(* CoDeSys 2.3.9.31 project: Test4(7Axis).pro *)
(* Libraries: STANDARD.LIB 5.6.98 11:03:02 *)

(* Task configuration *)
TASK Standard (PRIORITY := 0, INTERVAL := T#10ms);
	MAIN
END_TASK

(* Global variable list: Global_Variables *)
VAR_GLOBAL
(**DB Address**)
	DB8 AT %MW2010:ARRAY[0..100] OF INT;
(*******用到的数组值有以下变量*******)

	CigMakingSpeed  AT %IW330:INT;
(**Packer Address Define**)
	PackingSpeed  AT %IW332:INT;
(*ManPotentiometerSpeed  Address*)
	PotenSpeed AT %IW328:INT;
(*****Level Address  Define********)
	ElevatorLevel AT %IW324:INT;
(*****Drop Address  Define********)
	DropLevel AT %IW326:INT;

	Store_set_zero AT %MX1000.0 : BOOL;
	test_run AT %MX1000.6 : BOOL;
	StoreUnit_discharge_button AT %MX2603.6 : BOOL;
	Elevater_man_paikong AT %MX2603.7 :BOOL;
	test_run_unprotected AT %MX1000.7 : BOOL;
	test_maker_speed AT %MW1950 : INT;
	test_packer_speed AT %MW1952 : INT;
	Corner_manual_speed AT %MW254 : INT;
	Store_manual_speed AT %MW260 : INT;
	DropTrans_cig_speed AT %MW2320 : INT;(*下降口输送烟支速度*)(*******7Axis**********)
	DropTrans_speed_rpm AT %MW2340 : INT;(*下降口输送电机转速*)(******7Axis***********)


	Lift_p_parameter AT %MW270 : INT;
	Transfer_p_parameter AT %MW272 : INT;
	MakerExport_p_parameter AT %MW274 : INT;



	Emergency_stop AT %IX0.0:BOOL;(*紧急停止继电器*)
	MakerExit_power AT %IX0.1:BOOL;(*备用*)
	Sample_power AT %IX0.2:BOOL;(*取样伺服主电源*)
	Corner_power AT %IX0.3:BOOL;(*弯道伺服主电源*)
	Lift_power AT %IX0.4:BOOL;(*提升伺服主电源*)
	Transfer_power AT %IX0.5:BOOL;(*传送伺服主电源*)
	Slope_power AT %IX0.6:BOOL;(*斜向伺服主电源*)
	Store_power AT %IX0.7:BOOL;(*存储伺服主电源*)
	DropTrans_power AT %IX1.0:BOOL;(*下降口输送伺服主电源*)(****************************************************7Axis中用DropTrans_power替换原Spare10*************)

	Spare11 AT %IX1.1:BOOL;(*备用*)
	MakerExit_servo_fault AT %IX1.2:BOOL;(*备用*)
	Sample_servo_fault AT %IX1.3:BOOL;(*取样伺服控制器故障*)
	Corner_servo_fault AT %IX1.4:BOOL;(*弯道伺服控制器故障*)
	Lift_servo_fault AT %IX1.5:BOOL;(*提升伺服控制器故障*)
	Transfer_servo_fault AT %IX1.6:BOOL;(*传送伺服控制器故障*)
	Slope_servo_fault AT %IX1.7:BOOL;(*斜向伺服控制器故障*)
	Store_servo_fault AT %IX2.0:BOOL;(*存储伺服控制器故障*)
	DropTrans_servo_fault AT %IX2.1:BOOL;(*备用*)(********************************************************************7Axis中用DropTrans_servo_fault替换原Spare21*************)
	Spare22 AT %IX2.2:BOOL;(*备用*)
	Elevater_man_auto_sw AT %IX2.3:BOOL;(*备用*)
	Elevater_start_pb AT %IX2.4:BOOL;(*备用*)
	DropTransLowLevel AT %IX2.5:BOOL;(*下降口输送低料位*)(********************************************************7Axis中用DropTransLowLevel替换原Elevater_reset_pb*************)
	DropTransHighLevel AT %IX2.6:BOOL;(*下降口输送高料位*)(******************************************************7Axis中用DropTransHighLevel替换原Elevater_stop_pb*************)
	DropTransLimitLevel AT %IX2.7:BOOL;(*下降口输送极限料位*)(*****************************************************7Axis中用DropTransLimitLevel替换原Elevater_e_stop*************)
	Spare30 AT %IX3.0:BOOL;(*备用*)
	Spare31 AT %IX3.1:BOOL;(*备用*)
	MakerExit_sensor AT %IX3.2:BOOL;(*卷烟机出口有烟(备用)*)
	Sample_entrance_sensor AT %IX3.3:BOOL;(*取样入口有烟传感器*)
	Sample_entrance_jam_sensor AT %IX3.4:BOOL;(*取样入口堵塞传感器（备用）*)
	Corner_entrance_jam_sensor AT %IX3.5:BOOL;(*弯道入口堵塞传感器*)
	MakerExit_jam_sensor AT %IX3.6:BOOL;(*卷烟机出口堵塞（备用）*)
	Spare37 AT %IX3.7:BOOL;(*备用*)
	Downport_jam_sensor AT %IX4.0:BOOL;(*下降口堵塞传感器*)
	Slope_empty AT %IX4.1:BOOL;(*斜向通道空*)
	Transfer_cig_exist AT %IX4.2:BOOL;(*高架烟支传感器*)
	Transfer_overload_sensor AT %IX4.3:BOOL;(*传送过载传感器*)
	Spare44 AT %IX4.4:BOOL;(*备用*)
	Spare45 AT %IX4.5:BOOL;(*备用*)
	StoreUnit_e_stop_button :BOOL;
	Spare46 AT %IX4.6:BOOL;(*备用*)
	Spare47 AT %IX4.7:BOOL;(*备用*)
	Store_full AT %IX5.0:BOOL;(*存储器满传感器*)
	Store_empty AT %IX5.1:BOOL;(*存储器空传感器*)
	Store_overload AT %IX5.2:BOOL;(*存储器过载传感器*)
	Store_entrance_cig_exist AT %IX5.3:BOOL;(*存储器入口有烟传感器*)
	Store_entrance_jam AT %IX5.4:BOOL;(*存储器入口堵塞*)
	Store_overlimit AT %IX5.5:BOOL;(*存储器极限开关*)
	Store_running AT %IX5.6:BOOL;(*存储器运行中*)
	Store_enabled AT %IX5.7:BOOL;(*存储器使能*)
	sample_servo_enable_Q AT %QX4.0:BOOL;(*取样伺服驱动器使能*)
	Corner_servo_enable_Q AT %QX4.1:BOOL;(*弯道伺服驱动器使能*)
	Lift_servo_enable_Q AT %QX4.2:BOOL;(*提升伺服驱动器使能*)
	Transfer_servo_enable_Q AT %QX4.3:BOOL;(*传送伺服驱动器使能*)
	Slope_servo_enable_Q AT %QX4.4:BOOL;(*斜向伺服驱动器使能*)
	Store_servo_enable_Q AT %QX4.5:BOOL;(*存储伺服驱动器使能*)
	DropTrans_servo_enable_Q AT %QX4.6:BOOL;(*下降口输送伺服驱动器使能*)(*******************************7Axis中用DropTrans_servo_enable_Q替换原SpareOutput46*************)
	SpareOutput47 AT %QX4.7:BOOL;(*备用*)
	Elevater_start_Q AT %QX5.0:BOOL;(*备用*)
	Elevater_reset_Q AT %QX5.1:BOOL;(*备用*)
	Elevater_stop_Q AT %QX5.2:BOOL;(*备用*)
	Store_FaultReset_Q AT %QX5.3:BOOL;(*存储器故障复位*)
	Maker_enable_relay_Q AT %QX5.4:BOOL;(*卷烟机允许(备用)*)
	SpareOutput55 AT %QX5.5:BOOL;(*下降口急停复位*)
	SpareOutput56 AT %QX5.6:BOOL;(*备用*)
	Maker_QuickStop_Q AT %QX5.7:BOOL;(*卷烟机快停（备用）*)
	SpareOutput80 AT %QX8.0:BOOL;(*存储振动检测*)
	SpareOutput81 AT %QX8.1:BOOL;(*备用*)
	Packer_enable_relay_Q AT %QX8.2:BOOL;(*包装机允许（备用）*)
	Packer_LowSpeed_request_Q AT %QX8.3:BOOL;(*包装机低速请求（备用）*)
	SpareOutput84 AT %QX8.4:BOOL;(*备用*)
	SpareOutput85 AT %QX8.5:BOOL;(*系统主电源*)
	SpareOutput86 AT %QX8.6:BOOL;(*备用*)
	StoreUnit_start_Q AT %QX8.7:BOOL;(*备用*)
	StoreUnit_reset_Q AT %QX9.0:BOOL;(*备用*)
	StoreUnit_stop_Q AT %QX9.1:BOOL;(*备用*)
	SpareOutput92 AT %QX9.2:BOOL;(*备用*)
	SpareOutput93 AT %QX9.3:BOOL;(*备用*)
	SpareOutput94 AT %QX9.4:BOOL;(*备用*)
	SpareOutput95 AT %QX9.5:BOOL;(*备用*)
	SpareOutput96 AT %QX9.6:BOOL;(*备用*)
	SpareOutput97 AT %QX9.7:BOOL;(*备用*)


	DropTrans_servo_enable AT %MX3102.5:BOOL;(*下降口输送驱动器使能*)(*******************7Axis用*********************************)
	DropTrans_servo_initialized AT %MX3102.7:BOOL;(*下降口输送初始完成*)(*******************7Axis用*********************************)

	MakerExit_servo_enable AT %MX2102.5 : BOOL;
	MakerExit_servo_initialized AT %MX2102.7 : BOOL;
	sample_servo_enable AT %MX1502.5 : BOOL;
	sample_servo_initialized AT %MX1502.7 : BOOL;
	Corner_servo_enable AT %MX1602.5 : BOOL;
	Corner_servo_initialized AT %MX1602.7 : BOOL;
	Slope_servo_enable AT %MX1702.5 : BOOL;
	Slope_servo_initialized AT %MX1702.7 : BOOL;
	Store_servo_enable AT %MX1802.5 : BOOL;
	Lift_servo_enable AT %MX1902.5 : BOOL;
	Lift_servo_initialized AT %MX1902.7 : BOOL;
	Transfer_servo_enable AT %MX2002.5 : BOOL;
	Transfer_servo_initialized AT %MX2002.7 : BOOL;
	alarm_sample_entrance_jam AT %MX50.0 : BOOL;
	alarm_corner_entrance_jam AT %MX50.1 : BOOL;
	alarm_downport_entrance_jam AT %MX50.2 : BOOL;

	alarm_droptrans_jam AT %MX920.8 : BOOL;(*下降口输送堵塞*)(*******************7Axis用*********************************)



	alarm_transfer_overload AT %MX50.3 : BOOL;
	alarm_store_overload AT %MX50.4 : BOOL;
	alarm_store_entrance_jam AT %MX50.5 : BOOL;
	Elevater_manual_discharge AT %MX501.0 : BOOL;
	Elevater_auto_run AT %MX502.1 : BOOL;
	StoreUnit_man_run AT %MX550.1 : BOOL;
	StoreUnit_auto_run AT %MX552.1 : BOOL;
	StoreUnit_discharge_run AT %MX553.7 : BOOL;
	alarm_store_limit_on AT %MX60.2 : BOOL;
	alarm_store_full AT %MX71.2 : BOOL;
	alarm_encoder_fault AT %MX71.3 : BOOL;
	Maker_run AT %MX80.0 : BOOL;
	packer_run AT %MX80.1 : BOOL;
	MakerExit_servo_ethercat_fault AT %MX2600.0 : BOOL;
	Sample_servo_ethercat_fault AT %MX2600.1 : BOOL;
	Corner_servo_ethercat_fault AT %MX2600.2 : BOOL;
	Lift_servo_ethercat_fault AT %MX2600.3 : BOOL;
	Transfer_servo_ethercat_fault AT %MX2600.4 : BOOL;
	Slope_servo_ethercat_fault AT %MX2600.5 : BOOL;
	Store_servo_ethercat_fault AT %MX2600.6 : BOOL;
	DropTrans_servo_ethercat_fault AT %MX2600.7 : BOOL;(*下降口输送伺服通讯卡故障*)(*************************7Axis中用DropTrans_servo_ethercat_fault替换原Spare26007*************)
	Spare26010 AT %MX2601.0 : BOOL;
	Digital_Input1_ethercat_fault AT %MX2601.1 : BOOL;
	Digital_Input2_ethercat_fault AT %MX2601.2 : BOOL;
	Digital_Input3_ethercat_fault AT %MX2601.3 : BOOL;
	Digital_Input4_ethercat_fault AT %MX2601.4 : BOOL;
	Digital_Input5_ethercat_fault AT %MX2601.5 : BOOL;
	Digital_Input6_ethercat_fault AT %MX2601.6 : BOOL;
	Digital_Input7_ethercat_fault AT %MX2601.7 : BOOL;
	Digital_Output1_ethercat_fault AT %MX2602.0 : BOOL;
	Digital_Output2_ethercat_fault AT %MX2602.1 : BOOL;
	Digital_Output3_ethercat_fault AT %MX2602.2 : BOOL;
	Digital_Output4_ethercat_fault AT %MX2602.3 : BOOL;
	Analog_Input1_ethercat_fault AT %MX2602.4 : BOOL;
	Analog_Input2_ethercat_fault AT %MX2602.5 : BOOL;
	StoreUnit_Stop AT %MX2603.0 : BOOL;
	Elevater_Stop AT %MX2603.1 : BOOL;
	Manual_Run AT %MX2603.2 : BOOL;
	Auto_Run AT %MX2603.3 : BOOL;
	Elevater_Manual_Run AT %MX2603.4 : BOOL;
	test_run_light AT %MX1002.0 : BOOL;
	Downport_comp_output AT %MW1250 : INT;
	Maker_cig_speed AT %MW1300 : INT;
	Sample_cig_speed AT %MW1302 : INT;
	Corner_cig_speed AT %MW1304 : INT;
	Packer_cig_speed AT %MW1310 : INT;
	Life_cig_speed AT %MW1400 : INT;
	Transfer_cig_speed AT %MW1402 : INT;
	MakerExport_cig_speed AT %MW1404 : INT;
	MakerExport_speed_rpm AT %MW2236 : INT;
	Sample_speed_rpm AT %MW1536 : INT;
	Corner_speed_rpm AT %MW1636 : INT;
	Slope_speed_rpm AT %MW1736 : INT;
	Store_speed_rpm AT %MW1738 : INT;
	Corner_entrance_sensor_output AT %MW180 : INT;
	Downport_sensor_output AT %MW182 : INT;
	Store_CigNum AT %MW1880 : INT;
	Store_CigNum2 AT %MW1882 : INT;
	Store_cig_speed AT %MW1884 : INT;
	Slope_cig_speed AT %MW1886 : INT;
	Lift_speed_rpm AT %MW1936 : INT;
	Transfer_speed_rpm AT %MW2036 : INT;
	MakerExport_Servo_FaultNum AT %MW2800 : DWORD;
	Sample_Servo_FaultNum AT %MW2804 : DWORD;
	Corner_Servo_FaultNum AT %MW2808 : DWORD;
	Lift_Servo_FaultNum AT %MW2812 : DWORD;

	Transfer_Servo_FaultNum AT %MW2816 : DWORD;
	Slope_Servo_FaultNum AT %MW2820 : DWORD;
	Store_Servo_FaultNum AT %MW2824 : DWORD;
	DropTrans_Servo_FaultNum AT %MW2828 : DWORD;(*下降口输送伺服驱动器故障代码*)(***********7Axis增加下降口输送电机故障代码**************)




	Corner_pid_sp:INT;
	Corner_work_limit:INT;
	Corner_work_off_delay:INT;
	Corner_pid_p_gain:INT;
	Corner_p_parameter:INT;
	cig_dim:INT;
	Store_CigIn_Comp_speed1:INT;
	Store_CigIn_Comp_speed2:INT;
	Downport_CigIn_hight2:INT;
	Corner_pid_i_gain:INT;
	Maker_MaxSpeedLimit:INT;
	Packer_MaxSpeedLimit:INT;
	Store_empty_position:INT;
	Store_full_position:INT;
	Packer_LowSpeed_position:INT;
	Packer_enable_position:INT;
	Maker_stop_position:INT;
	Corner_entrance_hight_limit:INT;
	Corner_entrance_low_limt:INT;
	Downport_CigIn_hight1:INT;
	Corner_pid_deadband:INT;
	Downport_CigOut_hight1:INT;
	Downport_CigOut_hight2:INT;
	Store_CigOut_Comp_speed1:INT;
	Store_CigOut_Comp_speed2:INT;
	Downport_Highest_limit:INT;
	Downport_Lowest_limit:INT;
	Downport_CigIn_lowest_hight:INT;
	Corner_pid_output:INT;
	Corner_pid_pv:INT;
	DownPort_hight:INT;
	Store_percent:INT;
	Corner_lowlimit:INT;


	WriteFlag:BOOL;

END_VAR

(* POU MAIN, ST *)
PROGRAM MAIN
VAR
	aTON: TON;
	bTON: TON;
	Flag: BOOL := TRUE;
END_VAR
(*aTON(IN:=bTON.Q , PT:=T#200ms , Q=> , ET=> );
bTON(IN:= NOT aTON.Q , PT:=T#200ms , Q=> , ET=> );
Man_Auto_OP2:=bTON.Q;
*)

;

IF WriteFlag THEN

	DB8[0]:=Corner_pid_sp;
	DB8[36]:=Corner_work_limit;
	DB8[38]:=Corner_work_off_delay;
	DB8[4]:=Corner_pid_p_gain;
	DB8[40]:=Corner_p_parameter;
	DB8[46]:=cig_dim;
	DB8[52]:=Store_CigIn_Comp_speed1;
	DB8[54]:=Store_CigIn_Comp_speed2;
	DB8[56]:=Downport_CigIn_hight2;
	DB8[6]:=Corner_pid_i_gain;
	DB8[60]:=Maker_MaxSpeedLimit;
	DB8[62]:=Packer_MaxSpeedLimit;
	DB8[64]:=Store_empty_position;
	DB8[66]:=Store_full_position;
	DB8[68]:=Packer_LowSpeed_position;
	DB8[70]:=Packer_enable_position;
	DB8[72]:=Maker_stop_position;
	DB8[74]:=Corner_entrance_hight_limit;
	DB8[76]:=Corner_entrance_low_limt;
	DB8[78]:=Downport_CigIn_hight1;
	DB8[8]:=Corner_pid_deadband;
	DB8[80]:=Downport_CigOut_hight1;
	DB8[82]:=Downport_CigOut_hight2;
	DB8[84]:=Store_CigOut_Comp_speed1;
	DB8[86]:=Store_CigOut_Comp_speed2;
	DB8[88]:=Downport_Highest_limit;
	DB8[90]:=Downport_Lowest_limit;
	DB8[92]:=Downport_CigIn_lowest_hight;
	
	DB8[10]:=Corner_pid_output;
	DB8[2]:=Corner_pid_pv;
	DB8[26]:=DownPort_hight;
	DB8[50]:=Store_percent;

	DB8[58]:=Corner_lowlimit;

(*	WriteFlag:=0;*)
ELSE


	Corner_pid_sp:=DB8[0];
	Corner_work_limit:=DB8[36];
	Corner_work_off_delay:=DB8[38];
	Corner_pid_p_gain:=DB8[4];
	Corner_p_parameter:=DB8[40];
	cig_dim:=DB8[46];
	Store_CigIn_Comp_speed1:=DB8[52];
	Store_CigIn_Comp_speed2:=DB8[54];
	Downport_CigIn_hight2:=DB8[56];
	Corner_pid_i_gain:=DB8[6];
	Maker_MaxSpeedLimit:=DB8[60];
	Packer_MaxSpeedLimit:=DB8[62];
	Store_empty_position:=DB8[64];
	Store_full_position:=DB8[66];
	Packer_LowSpeed_position:=DB8[68];
	Packer_enable_position:=DB8[70];
	Maker_stop_position:=DB8[72];
	Corner_entrance_hight_limit:=DB8[74];
	Corner_entrance_low_limt:=DB8[76];
	Downport_CigIn_hight1:=DB8[78];
	Corner_pid_deadband:=DB8[8];
	Downport_CigOut_hight1:=DB8[80];
	Downport_CigOut_hight2:=DB8[82];
	Store_CigOut_Comp_speed1:=DB8[84];
	Store_CigOut_Comp_speed2:=DB8[86];
	Downport_Highest_limit:=DB8[88];
	Downport_Lowest_limit:=DB8[90];
	Downport_CigIn_lowest_hight:=DB8[92];
	
	Corner_pid_output:=DB8[10];
	Corner_pid_pv:=DB8[2];
	DownPort_hight:=DB8[26];
	Store_percent:=DB8[50];
	
	Corner_lowlimit:=DB8[58];

END_IF
END_PROGRAM
